// TIA Portal V20 export
FUNCTION_BLOCK "FB_PartPresenceCtrl"   // FB35, SCL
{ S7_Optimized_Access := 'TRUE' }
// stored: MemoryReserve 100, SetENOAutomatically false
   VAR_INPUT
      "iStart Control" : Bool;
      iMeasureValue : Real;
      iProdOK_LimHigh : Real;
      iProdOK_LimLow : Real;
      iProdMissing : Real;
   END_VAR
   VAR_OUTPUT
      oGoodPart : Bool;
      oBadpart : Bool;
   END_VAR
   VAR
      sRT_StartControl : R_TRIG;
      sBadPositioning { S7_SetPoint := 'True'} : Bool;
      sMissingBW { S7_SetPoint := 'True'} : Bool;
      sMissingPart : Bool;
      sStabilisationTime : TON_TIME;
   END_VAR
   VAR CONSTANT
      STABILISATION_TIME : Time := T#700ms;
   END_VAR
BEGIN
   REGION Description header 
       //==================================================================================
       // POSALUX Swiss SA / (C) Copyright 2025
       //----------------------------------------------------------------------------------
       // Title: CheckTimeout
       // Comment/Function: FB_PartPresenceCtrl
       //                   
       // Author: Fabien WALDT
       // Engineering: TIA Portal v19
       //----------------------------------------------------------------------------------
       // Change log table:
       // Version  | Date     | Expert in charge | Changes applied
       // ---------|----------|------------------|-----------------------------------------
       // 00.00.01 | 20250915 | WFA              | First released version
       // =================================================================================
   END_REGION

   REGION RT Start Cycle
       #sRT_StartControl(CLK := #"iStart Control");

      // IF #sRT_StartControl.Q THEN
       IF NOT #"iStart Control" THEN
           #oGoodPart := FALSE;
           #oBadpart := FALSE;
           #sBadPositioning := FALSE;
           #sMissingBW := FALSE;
           #sMissingPart := FALSE;
       END_IF;
   END_REGION

   REGION Stabilsation Time
       #sStabilisationTime(IN := #"iStart Control",
                           PT := #STABILISATION_TIME);
   END_REGION ;

   REGION Check Part
       IF #sStabilisationTime.Q THEN
           IF #iMeasureValue >= #iProdOK_LimLow AND #iMeasureValue <= #iProdOK_LimHigh THEN
               #oGoodPart := TRUE;
               #oBadpart := FALSE;
           ELSE
               #oGoodPart := FALSE;
               #oBadpart := TRUE;
               IF #iMeasureValue > #iProdOK_LimHigh THEN
                   #sBadPositioning := TRUE;
               ELSIF #iMeasureValue < #iProdMissing THEN
                   #sMissingPart := TRUE;
               ELSE
                   #sMissingBW := TRUE;
               END_IF;
           END_IF;
       END_IF;
   END_REGION
END_FUNCTION_BLOCK
